(* IEC 61131-3 sources: CodesysTest/alpha/export/Device.dev/Plc Logic/Application/FBs/DataHandlers/FB_ModbusDWORD.pou/HighWord.prop, 1 file *)

(* ---- Set.pm.st ---- *)
(*#-#-#-#-#-#-#-#-#-#---Declaration---#-#-#-#-#-#-#-#-#-#-#-#-#*)

VAR
END_VAR
(*#-#-#-#-#-#-#-#-#-#---Implementation---#-#-#-#-#-#-#-#-#-#-#-#-#*)

_highWord := HighWord;
